TYPE DriveOutputs :
STRUCT
	SetCounterValue : UDINT;
	TargetPosition : UDINT;
	TargetVelocity : INT;
	StartType : UINT;
	TargetAcceleration : UINT;
	TargetDeceleration : UINT;
END_STRUCT
END_TYPE

(* stored: Version 1.1.0.1, ProductVersion 3.1.4024.11
   DUT DriveOutputs: Id {e4a4846c-1480-4f4a-ac31-2b7ce5ceae8c} *)
